(* IEC 61131-3 sources: axcoderepos/test, 2 files *)

(* ---- test_fb.st ---- *)
USING Siemens.DemoMachine;
USING Siemens.DemoMachine.ConveyorUnit;
using  AxUnit;
NAMESPACE ConveyorTestFB

    {Test(start:=true)}
    FUNCTION PUBLIC TestConveyorMotorFB

        VAR_EXTERNAL
            //conveyor : ConveyorMotor;
            instConveyorMotor : ConveyorMotor;
                                                                                                                                                                                                                                                            //conveyor:Conveyor;
                                                                                                                                                                                                                                                        END_VAR

                                                                                                                                                                                                                                                        VAR_INPUT
                                                                                                                                                                                                                                                            start:bool;

        END_VAR
        VAR_TEMP
            res:bool;
        END_VAR

            instConveyorMotor(startStop:=start,outRun=>res);
            Assert.Equal(res,TRUE);

    END_FUNCTION
    {Test(start:=true,speed:=REAL#10.0)}
    FUNCTION PUBLIC TestConveyorDriveFB
        VAR_EXTERNAL
            instConveyorDrive : ConveyorDrive;
        END_VAR

        VAR_INPUT
            start:bool;
            speed:REAL;
        END_VAR
        VAR_TEMP
            run:bool;
            oSpeed:REAL;

        END_VAR

            instConveyorDrive(startStop:=start,speedSetpoint:=speed,outRun=>run,outSpeed=>oSpeed);
            Assert.Equal(run,FALSE);
            Assert.Equal(oSpeed,REAL#20.0);

    END_FUNCTION
END_NAMESPACE

(* ---- test_class.st ---- *)
USING AxUnit;
USING Siemens.DemoMachine;

NAMESPACE ConveyorTestClass

    {TestFixture}
    CLASS ConveyorMotorTest

        VAR PROTECTED
            conveyor : cConveyor;
            motor:cMotor;
            out:BOOL;
            in:BOOL;

        END_VAR

        {Test(btnStartStop:=TRUE)}
        METHOD PUBLIC MyTestMethod
            VAR_INPUT
                btnStartStop:BOOL;
            END_VAR

            motor.outRun:=REF(out);
            in:=btnStartStop;
            conveyor.startSop:=REF(in);
            conveyor.motor:=motor;
            conveyor.ConveyorControl();

            Assert.Equal(actual := out, expected := TRUE);

        END_METHOD
    END_CLASS

    {TestFixture}
    CLASS ConveyorDriveTest

        VAR PROTECTED
            conveyor : cConveyor;
            motor:cDriveMotor;
            out:BOOL;
            in:BOOL;
            outSpeed:REAL;
        END_VAR

        {Test(btnStartStop:=TRUE,setSpeed:=REAL#70.0)}
        METHOD PUBLIC MyTestMethod
            VAR_INPUT
                btnStartStop:BOOL;
                setSpeed:REAL;
            END_VAR

            motor.outRun:=REF(out);

            motor.outSpeed:=REF(outSpeed);
            in:=btnStartStop;
            conveyor.startSop:=REF(in);
            conveyor.motor:=motor;
            //set speed
            motor.SetSpeed(setSpeed);
            motor.outSpeed:=REF(outSpeed);
            //run/stop control
            conveyor.ConveyorControl();

            //Assert.Equal(actual := out, expected := btnStartStop);
            Assert.Equal(actual :=outSpeed, expected := REAL#60.0);

        END_METHOD
    END_CLASS
END_NAMESPACE
